PROGRAM Data_Shifting
VAR
	x, y			: 	INT ;
		
	testid			:	STRING := 'YI-10273';
//	testscanner		:	STRING := 'YI-10273';
	
	
END_VAR


IO.bBin_invi1 := (IO.abinID_Set[1] = '');
IO.bBin_invi2 := (IO.abinID_Set[2] = '');
IO.bBin_invi3 := (IO.abinID_Set[3] = '');
IO.bBin_invi4 := (IO.abinID_Set[4] = '');
IO.bBin_invi5 := (IO.abinID_Set[5] = '');
IO.bBin_invi6 := (IO.abinID_Set[6] = '');
IO.bBin_invi7 := (IO.abinID_Set[7] = '');
IO.bBin_invi8 := (IO.abinID_Set[8] = '');

IO.sbinID_Scanner := IO.sOutfeed_binID;

// ================================================  conv1
IF IO_Conveyor.bReceiving_Complete AND IO.abinID_Set[1] = '' THEN
	//IO.abinID_Set[1] := testid; 
	IO.abinID_Set[1] := IO.sReceiving_binID;
END_IF 

IF IO_Logs.bConv1_Out.Q THEN
	IF (IO.abinID_Set[1] <> '') AND (IO.abinID_Set[2] = '') THEN
		IO.abinID_Set[2] := IO.abinID_Set[1];
		IO.abinID_Set[1] := '' ;
	END_IF
END_IF

// ================================================  conv2
IF IO_Logs.bConv2_In.Q THEN
	IF (IO.abinID_Set[2] <> '') AND (IO.abinID_Set[3] = '') THEN
		IO.abinID_Set[3] := IO.abinID_Set[2];
		IO.abinID_Set[2] := '' ;
	END_IF
END_IF

IF IO_Logs.bConv2_Out.Q THEN
	IF (IO.abinID_Set[3] <> '') AND (IO.abinID_Set[4] = '') THEN
		IO.abinID_Set[4] := IO.abinID_Set[3];
		IO.abinID_Set[3] := '' ;
	END_IF
END_IF

// ================================================  conv3
IF IO_Logs.bConv3_In.Q THEN
	IF (IO.abinID_Set[4] <> '') AND (IO.abinID_Set[5] = '') THEN
		IO.abinID_Set[5] := IO.abinID_Set[4];
		IO.abinID_Set[4] := '' ;
	END_IF
END_IF

IF IO_Logs.bConv3_Out.Q THEN
	IF (IO.abinID_Set[5] <> '') AND (IO.abinID_Set[6] = '') THEN
		IO.abinID_Set[6] := IO.abinID_Set[5];
		IO.abinID_Set[5] := '' ;
	END_IF
END_IF

// ================================================  conv4
IF IO_Logs.bConv4_In.Q THEN
	IF (IO.abinID_Set[6] <> '') AND (IO.abinID_Set[7] = '') THEN
		IO.abinID_Set[7] := IO.abinID_Set[6];
		IO.abinID_Set[6] := '' ;
	END_IF
END_IF

IF IO_Logs.bConv4_Out.Q THEN
	IF (IO.abinID_Set[7] <> '') AND (IO.abinID_Set[8] = '') THEN
		IO.abinID_Set[8] := IO.abinID_Set[7];
		IO.abinID_Set[7] := '' ;
	END_IF
	
	IF IO.abinID_Set[8] = IO.sbinID_Scanner THEN
		IO.abinID_Set[8] := '' ;
	END_IF
END_IF

END_PROGRAM

(* stored: Version 1.1.0.1, ProductVersion 3.1.4024.12
   POU Data_Shifting: Id {3c954cfc-5714-4c36-8a0c-c978ca237666}, SpecialFunc None *)
